# B&R Automation Studio project laba_3BR-master
Automation Studio 4.5.2.102

## Logical view

### Global.var - Global variables
```iecst
VAR
	AxisX : ACP10AXIS_typ := (0);
	AxisX_EncIf : SdcEncIf16_typ := (0);
	AxisX_DrvIf : SdcDrvIf16_typ := (0);
	AxisX_DiDoIf : SdcDiDoIf_typ := (0);
	AxisX_HW : SdcHwCfg_typ := (0);
	gAxis01 : ACP10AXIS_typ := (0);
	gAxis02 : ACP10AXIS_typ := (0);
	gAxisTest : ACP10AXIS_typ := (0);
	gAxisTest_HW : SdcHwCfg_typ := (0);
	gAxisTest_DrvIf : SdcDrvIf16_typ := (0);
	gAxisTest_DiDoIf : SdcDiDoIf_typ := (0);
	gAxisTest_ModuleOk : BOOL := 0;
	gAxis03 : ACP10AXIS_typ := (0);
	gAxis03_HW : SdcHwCfg_typ := (0);
	gAxis03_DrvIf : SdcDrvIf16_typ := (0);
	gAxis03_DiDoIf : SdcDiDoIf_typ := (0);
	gAxis03_ModuleOk : BOOL := 0;
	CNCsys : ARNC0CNC_typ;
	gAxis04 : ACP10AXIS_typ := (0);
	gAxis05 : ACP10AXIS_typ := (0);
	gAxis05_HW : SdcHwCfg_typ := (0);
	gAxis05_DrvIf : SdcDrvIf16_typ := (0);
	gAxis05_EncIf1 : SdcEncIf16_typ := (0);
	gAxis05_DiDoIf : SdcDiDoIf_typ := (0);
	gAxis05_MotorStep0 : INT := 0;
	coil_powered : BOOL := FALSE;
	coil_pwm_value : INT := 0;
	fb_regulator : FB_Regulator;
	pwm_period : UINT := 0;
	axis_X : FB_Axis := (0);
	iPosHwEnd : BOOL := FALSE;
	iNegHwEnd : BOOL := FALSE;
	iActPos : USINT := 0;
	oSetPos : USINT := 0;
END_VAR
```

### Package Logical/gAxis03obj - gAxis03obj

### gAxis03i.ax
```
InitParameter (Version=3.13.1, NcSwId=Acp10)
  ACP10AXIS_typ:
    dig_in:
      level:
        reference = ncACTIV_HI
        pos_hw_end = ncACTIV_HI
        neg_hw_end = ncACTIV_HI
        trigger1 = ncACTIV_HI
        trigger2 = ncACTIV_HI
    encoder_if:
      parameter:
        count_dir = ncSTANDARD
        scaling:
          load:
            units = 1000
            rev_motor = 1
    limit:
      parameter:
        v_pos = 10000
        v_neg = 10000
        a1_pos = 50000
        a2_pos = 50000
        a1_neg = 50000
        a2_neg = 50000
        t_jolt = 0
        t_in_pos = 0
        pos_sw_end = 2000000000
        neg_sw_end = -2000000000
        ds_warning = 500
        ds_stop = 1000
        a_stop = 1.0e30
        dv_stop = 0
        dv_stop_mode = ncOFF
    controller:
      mode = ncPOSITION
      position:
        kv = 50
        tn = 0
        t_predict = 0.01
        t_total = 0.01
        p_max = 1.0e30
        i_max = 0
      speed:
        kv = 2.0
        tn = 0
        t_filter = 0.0
        isq_filter1:
          type = ncOFF
          a0 = 0.0
          a1 = 0.0
          b0 = 0.0
          b1 = 0.0
          b2 = 0.0
          c0_par_id = 0
          c1_par_id = 0
        isq_filter2:
          type = ncOFF
          a0 = 0.0
          a1 = 0.0
          b0 = 0.0
          b1 = 0.0
          b2 = 0.0
          c0_par_id = 0
          c1_par_id = 0
        isq_filter3:
          type = ncOFF
          a0 = 0.0
          a1 = 0.0
          b0 = 0.0
          b1 = 0.0
          b2 = 0.0
          c0_par_id = 0
          c1_par_id = 0
      uf:
        type = ncLINEAR
        auto_config = ncMOTOR_PAR
        u0 = 0
        un = 0
        fn = 50.0
        k_f_slip = 0
      ff:
        torque_load = 0.0
        torque_pos = 0.0
        torque_neg = 0.0
        kv_torque = 0.0
        inertia = 0.0
        t_filter_a = 0.0
    move:
      stop:
        parameter[0]:
          decel_ramp = ncA_LIMIT
          controller = ncON
        parameter[1]:
          decel_ramp = ncA_LIMIT
          controller = ncON
        parameter[2]:
          decel_ramp = ncA_LIMIT
          controller = ncON
        parameter[3]:
          decel_ramp = ncA_LIMIT
          controller = ncON
        quickstop:
          decel_ramp = ncA_LIMIT
        drive_error:
          decel_ramp = ncA_LIMIT
      homing:
        parameter:
          s = 0
          v_switch = 5000
          v_trigger = 500
          a = 50000
          mode = ncEND_SWITCH
          edge_sw = ncPOSITIVE
          start_dir = ncPOSITIVE
          trigg_dir = ncPOSITIVE
          ref_pulse = ncOFF
          fix_dir = ncOFF
          tr_s_block = 0
          torque_lim = 0
          ds_block = 0
          ds_stop = 0
      basis:
        parameter:
          v_pos = 5000
          v_neg = 5000
          a1_pos = 50000
          a2_pos = 50000
          a1_neg = 50000
          a2_neg = 50000
    message:
      text:
        parameter:
          format = ncBREAK
          columns = 80
          data_modul = acp10etxen
```

### Program Logical/SDCAxisCtrl_X (ANSIC)

#### Variables.var
```iecst
VAR
	min_task : INT := 7000;
	desired_speed : INT := 0;
	axis_X : FB_Axis;
	coil_powered : BOOL := FALSE;
	coil_pwm_value : {REDUND_UNREPLICABLE} INT := 200;
	fb_controller : FB_Controller;
	pwm_period : {REDUND_UNREPLICABLE} UINT := 200;
	Already_Homed : BOOL := FALSE;
	k : INT := 0;
	reset : BOOL := FALSE;
END_VAR
```

#### Main.c
```c
#include <bur/plctypes.h>

#ifdef _DEFAULT_INCLUDES
	#include <AsDefault.h>
#endif

void increase_counters(void);
void Homing(void);

void _INIT ProgramInit(void)
{
	//Устанваливаем типы SDC модулей
	AxisX_HW.EncIf1_Typ = ncSDC_ENC16;
	AxisX_HW.DiDoIf_Typ = ncSDC_DIDO;
	AxisX_HW.DrvIf_Typ = ncSDC_DRVSERVO16;

	//Устанавливаем имена переменных
	strcpy(AxisX_HW.EncIf1_Name, "AxisX_EncIf");
	strcpy(AxisX_HW.DrvIf_Name, "AxisX_DrvIf");
	strcpy(AxisX_HW.DiDoIf_Name, "AxisX_DiDoIf");

	//Устанавливаем входы готовности и нормальной работы
	AxisX_EncIf.iEncOK = 1;
	AxisX_DrvIf.iDrvOK = 1;
	AxisX_DrvIf.iStatusEnable = 1;
	AxisX_DiDoIf.iDriveReady = 1;

	fb_regulator.dt = 0.002;
	fb_regulator.k_i = 0.16;
	fb_regulator.k_p = 0.0064;
	fb_regulator.max_abc_value = 24.0;

	pwm_period = 200;
}

void _CYCLIC ProgramCyclic(void)
{
	increase_counters();
	AxisX_EncIf.iActTime = (INT)AsIOTimeCyclicStart();
	AxisX_DiDoIf.iPosHwEnd = axis_X.endswitch_a_reached;
	AxisX_DiDoIf.iNegHwEnd = axis_X.endswitch_b_reached;

	if(coil_powered == 1)
	{
		/*if(!Already_Homed)
		{
			Homing();
		}
		else
		{*/
			increase_counters();
			axis_X.reset_counter = 0;
			FB_Axis(&axis_X);
			coil_pwm_value = 32767;
		AxisX_DiDoIf.iPosHwEnd = axis_X.endswitch_a_reached;
		AxisX_DiDoIf.iNegHwEnd = axis_X.endswitch_b_reached;
			FB_Axis(&axis_X);

			fb_regulator.e = (AxisX_DrvIf.oSetPos*100)  - axis_X.speed;//oSetPos;
			FB_Regulator(&fb_regulator);

			axis_X.u = fb_regulator.u ;
			FB_Axis(&axis_X);//}
	}
	else
	{
		coil_pwm_value = 0;
		fb_regulator.e = 0 ;
		FB_Regulator(&fb_regulator);
		axis_X.u = 0;
		FB_Axis(&axis_X);

	}
	// COUNTER1 = axis_X.counter

	//COUNTER2 += axis_X.counter - COUNTER1;
}

void increase_counters(void)
{
	AxisX_EncIf.iLifeCnt++;
	AxisX_DiDoIf.iLifeCntDriveEnable++;
	AxisX_DiDoIf.iLifeCntDriveReady++;
	AxisX_DiDoIf.iLifeCntNegHwEnd++;
	AxisX_DiDoIf.iLifeCntPosHwEnd++;
	AxisX_DiDoIf.iLifeCntReference++;
	AxisX_DrvIf.iLifeCnt++;
}

void Homing(void)
{
	increase_counters();
	coil_pwm_value = 32767;
	iPosHwEnd = axis_X.endswitch_a_reached;
	iNegHwEnd = axis_X.endswitch_b_reached;
	FB_Axis(&axis_X);

	fb_regulator.e = (AxisX_DrvIf.oSetPos * 10) - axis_X.speed;//oSetPos;
	FB_Regulator(&fb_regulator);

	axis_X.u = fb_regulator.u ;
	FB_Axis(&axis_X);
	if (iPosHwEnd)
	{
		coil_pwm_value = 0;
		fb_regulator.e = 0;
		FB_Regulator(&fb_regulator);
		axis_X.u = 0;
		FB_Axis(&axis_X);
		axis_X.reset_counter = 1;
		FB_Axis(&axis_X);
		if(k == 200)
		{
			Already_Homed = 1;
			FB_Axis(&axis_X);
		}
		k++;

	}

}

void _EXIT ProgramExit(void)
{
	// Insert code here

}
```

Listed in the project but not available here: Logical/Global.typ, Logical/Libraries, Logical/AxisApt, Logical/Types.typ, Logical/AxisInit, Logical/acp10etxen, Logical/ncsdcctrl, Logical/gAxis05obj
